Omron CX-Programmer project NewProject (CX-Programmer 9.61)

# PLC NewPLC1: CP1E E20

## Global symbols (name address type ; comment)
0.00 BOOL  ; UP1
0.01 BOOL  ; UP2
0.02 BOOL  ; RESET
10.00 BOOL  ; LAMPU1
10.01 BOOL  ; L2
10.02 BOOL  ; L3

## Program NewProgram1 (cyclic task 0)
Local symbols
U CHANNEL
o 100.00 BOOL

### Section Section1

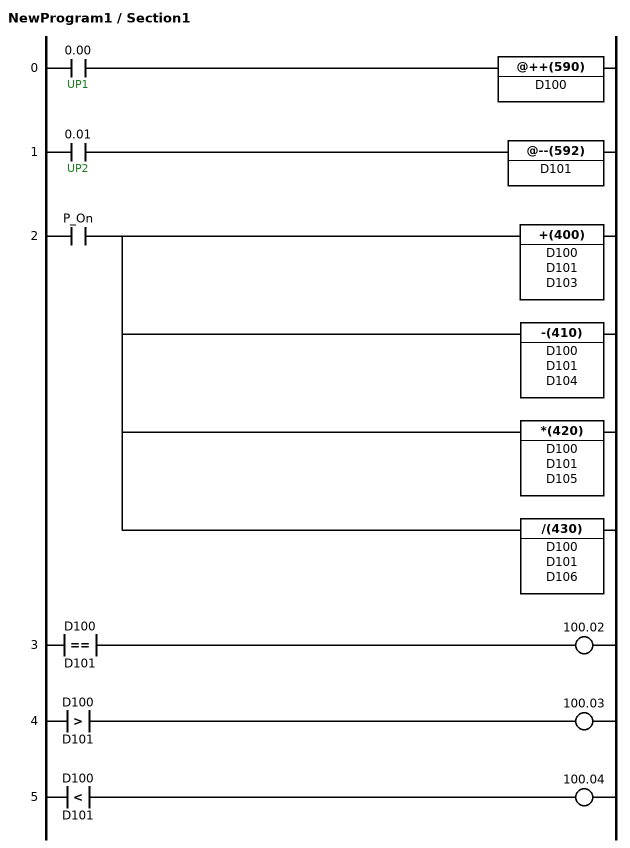
; rung 0
LD 0.00  ; UP1
@++(590) D100
; rung 1
LD 0.01  ; UP2
@--(592) D101
; rung 2
LD P_On
+(400) D100 D101 D103
-(410) D100 D101 D104
*(420) D100 D101 D105
/(430) D100 D101 D106
; rung 3
LD=(300) D100 D101
OUT 100.02
; rung 4
LD>(320) D100 D101
OUT 100.03
; rung 5
LD<(310) D100 D101
OUT 100.04

### Section END
; rung 0
END(001)